FUNCTION_BLOCK CROSSCOMM_PEER_16697678DCF9C13D3 (* Service Interface Function Block Type *)
  (* Standard: 61499-2 *)
  (* Version 0.0, 9/22/2017, bababen, nxtControl GmbH, template *)
  PACKAGE Main;
  (* Compiler Cpp nxtControl builtin 1.0 *)
  {SET_ATTRIBUTE(Runtime.FBType.ImplementingType, Runtime.System#DYNGEN_CROSSCOMM_PEER)}
  {SET_ATTRIBUTE(Configuration.GenericFBType.InterfaceParams, Runtime.System#<InterfaceList> <EventOutputs> <Event Name="PUSHED" /> </EventOutputs> <OutputVars /> </InterfaceList>)}
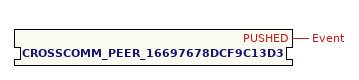
  EVENT_OUTPUT
    PUSHED;
  END_EVENT
  EC_STATES
    START;
  END_STATES
END_FUNCTION_BLOCK
